Fanuc KAREL source: ko00150.KL

-- PROVISIONAL review KL for V1013-1; original PC SHA256 b569970c565c63945857dafd11a12b6c664f2cc4d121c6dec3941c685162e85d
-- Incomplete behavior may be omitted. Consult companion uncertainty JSON. Do not deploy.
PROGRAM KO00150
%NOLOCKGROUP
VAR
  R : REAL
  N : REAL
-- UNRESOLVED_DECL CFG type=00001c
-- UNRESOLVED_DECL OUT type=000102
BEGIN
  -- UNRESOLVED_PC offsets 5-13; opcodes 9D,64,23
  -- UNRESOLVED_PC offsets 18-29; opcodes 2E,23
  -- UNRESOLVED_PC offsets 34-44; opcodes 9D,22,A5
  -- UNRESOLVED_PC offsets 49-106; opcodes 27,22,22,22,22,22,22,22,76,7E,4A
  -- UNRESOLVED_PC offsets 111-115; opcodes 7F
END KO00150
